(* IEC 61131-3 sources: RL_MAR/experiments/comparison/autoplc/results/gpt-4o_20260511_211137/med_30, 1 file *)

(* ---- med_30_1.st ---- *)
FUNCTION_BLOCK MuseumClimateControl
VAR_INPUT
    HumiditySensor : REAL;
    TemperatureSensor : REAL;
    LightSensor : BOOL;
END_VAR

VAR_OUTPUT
    HVACSystem : BOOL;
    Humidifier : BOOL;
    Dehumidifier : BOOL;
    LightControl : BOOL;
END_VAR

VAR
    TargetHumidity : REAL := 50.0;
    TargetTemperature : REAL := 20.0;
    LightThreshold : BOOL := TRUE;
END_VAR

// Implementing the control logic for the museum climate control system
// Humidity Control Logic
IF HumiditySensor < TargetHumidity THEN
    Humidifier := TRUE;
    Dehumidifier := FALSE;
ELSIF HumiditySensor > TargetHumidity THEN
    Humidifier := FALSE;
    Dehumidifier := TRUE;
ELSE
    Humidifier := FALSE;
    Dehumidifier := FALSE;
END_IF

// Temperature Control Logic
IF TemperatureSensor < TargetTemperature OR TemperatureSensor > TargetTemperature THEN
    HVACSystem := TRUE;
ELSE
    HVACSystem := FALSE;
END_IF

// Lighting Control Logic
IF LightSensor = TRUE AND LightThreshold = TRUE THEN
    LightControl := FALSE;
ELSE
    LightControl := TRUE;
END_IF

END_FUNCTION_BLOCK
